// TIA Portal project "Three Motors in PLC with Delayed ON and OFF Time Program" (V17)
// Three Motors in PLC with Delayed ON and OFF Time Program
// When Switch is ON,
// After 5s, Motor 1 will be ON
// After 10s, Motor 2 will be ON
// After 15s, Motor 3 will be ON
// After 20s, all the Motors will be OFF

(* hardware
DEVICE "S7-1200 station_1"  S7-1200 Station
   slot 0: "Rack_0"  S7-1200 Rack  Rack  V1.0
   slot 1: "PLC_1"  CPU 1211C AC/DC/Rly  6ES7 211-1BE40-0XB0  V4.5
*)

// ===== PLC "PLC_1"  CPU 1211C AC/DC/Rly =====

VAR_GLOBAL   // PLC tag table "Default tag table"
   "PB Switch" AT %I0.0 : Bool;
   "Motor 1" AT %Q0.0 : Bool;
   "Motor 2" AT %Q0.1 : Bool;
   "Motor 3" AT %Q0.2 : Bool;
   "Tag_1" AT %M0.0 : Bool;
END_VAR

// folder: System blocks/Program resources

DATA_BLOCK "IEC_Timer_0_DB"   // DB1
{ S7_Optimized_Access := 'TRUE' }
AUTHOR : Simatic
FAMILY : IEC
NAME : IEC_TMR
VERSION : 1.0
// stored: InstanceOfName IEC_TIMER
"IEC_TIMER"
BEGIN
END_DATA_BLOCK

DATA_BLOCK "IEC_Timer_0_DB_4"   // DB5
{ S7_Optimized_Access := 'TRUE' }
AUTHOR : Simatic
FAMILY : IEC
NAME : IEC_TMR
VERSION : 1.0
// stored: InstanceOfName IEC_TIMER
"IEC_TIMER"
BEGIN
END_DATA_BLOCK

DATA_BLOCK "IEC_Timer_0_DB_5"   // DB6
{ S7_Optimized_Access := 'TRUE' }
AUTHOR : Simatic
FAMILY : IEC
NAME : IEC_TMR
VERSION : 1.0
// stored: InstanceOfName IEC_TIMER
"IEC_TIMER"
BEGIN
END_DATA_BLOCK

DATA_BLOCK "IEC_Timer_0_DB_6"   // DB7
{ S7_Optimized_Access := 'TRUE' }
AUTHOR : Simatic
FAMILY : IEC
NAME : IEC_TMR
VERSION : 1.0
// stored: InstanceOfName IEC_TIMER
"IEC_TIMER"
BEGIN
END_DATA_BLOCK

// folder: (top level)

ORGANIZATION_BLOCK "Main"   // OB1, LAD, ProgramCycle
TITLE = "Main Program Sweep (Cycle)"
{ S7_Optimized_Access := 'TRUE' }
VERSION : 0.1
   VAR_INPUT
      Initial_Call : Bool;   // Initial call of this OB
      Remanence : Bool;   // =True, if remanent data are available
   END_VAR
BEGIN

REGION Network 1
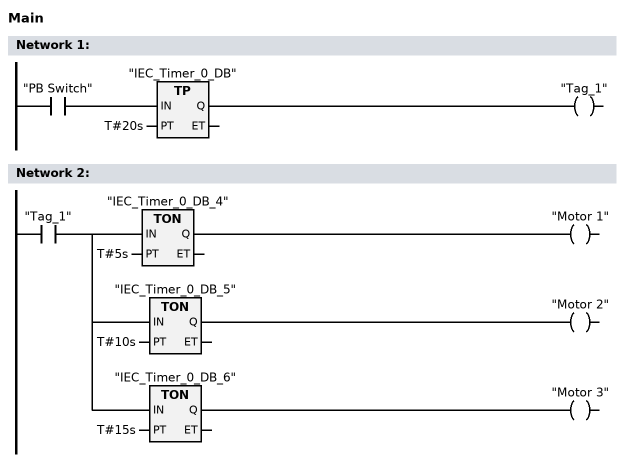
   "IEC_Timer_0_DB".TP(IN := "PB Switch", PT := T#20s);
   "Tag_1" := "IEC_Timer_0_DB".Q;
END_REGION

REGION Network 2
   "IEC_Timer_0_DB_4".TON(IN := "Tag_1", PT := T#5s);
   "Motor 1" := "IEC_Timer_0_DB_4".Q;
   "IEC_Timer_0_DB_5".TON(IN := "Tag_1", PT := T#10s);
   "Motor 2" := "IEC_Timer_0_DB_5".Q;
   "IEC_Timer_0_DB_6".TON(IN := "Tag_1", PT := T#15s);
   "Motor 3" := "IEC_Timer_0_DB_6".Q;
END_REGION
END_ORGANIZATION_BLOCK